// TIA Portal V18 export
// export: Created 2026-03-12T16:04:33.8604077Z, ExportSetting WithDefaults, DisplayName Totally Integrated Automation Portal, DisplayVersion V18 Update 5, DisplayName TIA Portal Openness, DisplayVersion V18 Update 5, DisplayName TIA Portal Version Control Interface, DisplayVersion V18, DisplayName SINAMICS Startdrive Advanced, DisplayVersion V18, DisplayName SINAMICS Startdrive G130, G150, S120, S150, SINAMICS MV, S210, DisplayVersion V18, DisplayName SINAMICS Startdrive G110M, G120, G120C, G120D, G120P, G115D, DisplayVersion V18, DisplayName STEP 7 Professional, DisplayVersion V18 Update 5, DisplayName STEP 7 Safety, DisplayVersion V18, DisplayName WinCC Professional, DisplayVersion V18 Update 5
FUNCTION_BLOCK "FB BITS TO WORD"   // FB4, SCL
{ S7_Optimized_Access := 'TRUE' }
VERSION : 0.1
// stored: AutoNumber true, IsIECCheckEnabled false, IsRetainMemResEnabled false, MemoryReserve 100, SetENOAutomatically false, UDAEnableTagReadback false
   VAR_INPUT
      SIGNAL_Bit0 : Bool;   // Sinal de entrada 1
      SIGNAL_Bit1 : Bool;   // Sinal de entrada 2
      SIGNAL_Bit2 : Bool;   // Sinal de entrada 3
      SIGNAL_Bit3 : Bool;   // Sinal de entrada 4
      SIGNAL_Bit4 : Bool;   // Sinal de entrada 5
      SIGNAL_Bit5 : Bool;   // Sinal de entrada 6
      SIGNAL_Bit6 : Bool;   // Sinal de entrada 7
      SIGNAL_Bit7 : Bool;   // Sinal de entrada 8
      SIGNAL_Bit8 : Bool;   // Sinal de entrada 9
      SIGNAL_Bit9 : Bool;   // Sinal de entrada 10
      SIGNAL_Bit10 : Bool;   // Sinal de entrada 11
      SIGNAL_Bit11 : Bool;   // Sinal de entrada 12
      SIGNAL_Bit12 : Bool;   // Sinal de entrada 13
      SIGNAL_Bit13 : Bool;   // Sinal de entrada 14
      SIGNAL_Bit14 : Bool;   // Sinal de entrada 15
      SIGNAL_Bit15 : Bool;   // Sinal de entrada 16
   END_VAR
   VAR_OUTPUT
      BITS_TO_WORD : Word;   // Word de saída com os sinais montados
   END_VAR
BEGIN
   // Word Alarmes - Montando bits em uma word

   // Bits recebidos de campo
   #"BITS_TO_WORD".%X0 := #SIGNAL_Bit0;
   #"BITS_TO_WORD".%X1 := #SIGNAL_Bit1;
   #"BITS_TO_WORD".%X2 := #SIGNAL_Bit2;
   #"BITS_TO_WORD".%X3 := #SIGNAL_Bit3;
   #"BITS_TO_WORD".%X4 := #SIGNAL_Bit4;
   #"BITS_TO_WORD".%X5 := #SIGNAL_Bit5;
   #"BITS_TO_WORD".%X6 := #SIGNAL_Bit6;
   #"BITS_TO_WORD".%X7 := #SIGNAL_Bit7;
   #"BITS_TO_WORD".%X8 := #SIGNAL_Bit8;
   #"BITS_TO_WORD".%X9 := #SIGNAL_Bit9;
   #"BITS_TO_WORD".%X10 := #SIGNAL_Bit10;
   #"BITS_TO_WORD".%X11 := #SIGNAL_Bit11;
   #"BITS_TO_WORD".%X12 := #SIGNAL_Bit12;
   #"BITS_TO_WORD".%X13 := #SIGNAL_Bit13;
   #"BITS_TO_WORD".%X14 := #SIGNAL_Bit14;
   #"BITS_TO_WORD".%X15 := #SIGNAL_Bit15;
END_FUNCTION_BLOCK
